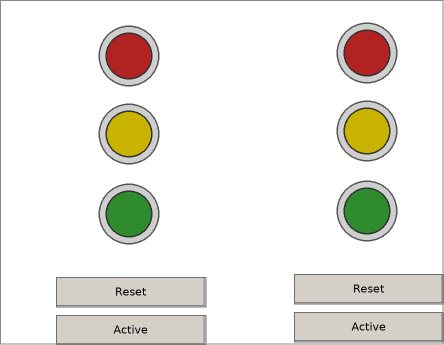
VISUALIZATION TrafficLight  // 444x345
    Lamp1 (94,21 70x70), variable: GVL_HMI_TrafficLight.LED_Red, style: Lamp-Lamp1-Red
    Lamp1 (94,99 70x70), variable: GVL_HMI_TrafficLight.LED_Yellow, style: Lamp-Lamp1-Yellow
    Lamp1 (94,179 70x70), variable: GVL_HMI_TrafficLight.LED_Green, style: Lamp-Lamp1-Green
    Button (56,277 150x30), "Reset"
        tap GVL_HMI_TrafficLight.btnReset
    Button (56,315 150x30), "Active"
        tap GVL_HMI_TrafficLight.btnActive
    Lamp1 (332,18 70x70), variable: GVL_HMI_TrafficLight.LED_Red_1, style: Lamp-Lamp1-Red
    Lamp1 (332,96 70x70), variable: GVL_HMI_TrafficLight.LED_Yellow_1, style: Lamp-Lamp1-Yellow
    Lamp1 (332,176 70x70), variable: GVL_HMI_TrafficLight.LED_Green_1, style: Lamp-Lamp1-Green
    Button (294,274 150x30), "Reset"
        tap GVL_HMI_TrafficLight.btnReset_1
    Button (294,312 150x30), "Active"
        tap GVL_HMI_TrafficLight.btnActive_1
END_VISUALIZATION

(* stored: Version 1.1.0.1, ProductVersion 3.1.4024.12
   Visu TrafficLight: Id {47e57637-d8a3-405f-bebf-f3fc73924987} *)
